{attribute 'enable_dynamic_creation'}
FUNCTION_BLOCK FB_Cartridge EXTENDS FB_PieceBase
VAR_INPUT
END_VAR
VAR_OUTPUT
END_VAR
VAR
END_VAR

METHOD FB_init : BOOL
VAR_INPUT
	bInitRetains : BOOL; // if TRUE, the retain variables are initialized (warm start / cold start)
	bInCopyCode : BOOL;  // if TRUE, the instance afterwards gets moved into the copy code (online change)
END_VAR
eObjectType := E_ObjectType.OBJECTTYPE_Cartridge;
eObjectGroup := E_ObjectGroup.OBJECTGROUP_Piece;
END_METHOD

END_FUNCTION_BLOCK

(* stored: Version 1.1.0.1, ProductVersion 3.1.4022.18
   POU FB_Cartridge: Id {b5a93d8b-1f56-4962-aae7-5107faba618a}, SpecialFunc None
   Method FB_init: Id {643afb72-2420-4c09-9525-1f178a1636d0} *)
